{attribute 'GeneratedUsingTerminal: EL9221-4030-0018'}
{attribute addProperty BoxType "EL9221-4030-0018"}
{attribute addProperty Id "OCP_InputsAT %I*OCP_Inputs_8CCE65FB11OCP_OutputsAT %Q*OCP_Outputs_010149342WcStateAT %I*WcState_9091E0EB2InfoDataAT %I*InfoData_32EB74EA10"}
{attribute addProperty CRC "2183379159"}
{attribute addProperty Size "25"}
TYPE EL9221_8223B8D7 EXTENDS EtcSlaveTerminalBase_947E5A46 :
STRUCT
	{attribute addProperty Name "OCP_Inputs"}
	OCP_Inputs : OCP_Inputs_8CCE65FB;
	{attribute addProperty Name "OCP_Outputs"}
	OCP_Outputs : OCP_Outputs_01014934;
	{attribute addProperty Name "WcState"}
	WcState : WcState_9091E0EB;
	{attribute addProperty Name "InfoData"}
	InfoData : InfoData_32EB74EA;
END_STRUCT
END_TYPE

(* stored: Version 1.2.0.0, ProductVersion 3.1.4024.9
   DUT EL9221_8223B8D7: Id {de2dcf0c-f159-4f77-acb6-238ea6ff2bfa} *)
